FUNCTION_BLOCK EL4004
VAR
	_io : EL4xx4_Data;
	{attribute addProperty Name "WcState"}
	_wcState : WcStateBase;
	{attribute addProperty Name "Info data"}
	_infoData : InfoDataAds;
END_VAR

PROPERTY IO : REFERENCE TO EL4xx4_Data
GET
IO REF= _io;
END_GET
END_PROPERTY

PROPERTY WcState : REFERENCE TO WcStateBase
GET
WcState REF= _wcState;
END_GET
END_PROPERTY

END_FUNCTION_BLOCK

(* stored: Version 1.1.0.1, ProductVersion 3.1.4024.9
   POU EL4004: Id {c0b564fe-ec29-0880-162f-51f61c40f883}, SpecialFunc None
   Property IO: Id {ab38dcf8-4efe-0b7f-1dee-6c95edb34fa0}
   Get Get: Id {befb17e9-0b1c-00cf-2d17-64bd2d70259f}
   Property WcState: Id {b931cec5-9254-06af-283e-108fb84dd794}
   Get Get: Id {f729aad8-2ed1-0ba5-262c-54aba0f0d031} *)
